{attribute addProperty BoxType "EPP1816-3008-0016"}
{attribute addProperty Id "StatusAT %I*Status_9EB472D91620ValueAT %I*INT16217"}
{attribute addProperty CRC "911372288"}
{attribute addProperty SizeInBites "32"}
{attribute addProperty SizeInBytes "4"}
TYPE AI_Inputs_Channel_36527000 :
STRUCT
	{attribute addProperty Name "Status"}
	Status AT %I* : Status_9EB472D9;
	{attribute addProperty Name "Value"}
	Value AT %I* : INT;
END_STRUCT
END_TYPE

(* stored: Version 1.2.0.0, ProductVersion 3.1.4024.9
   DUT AI_Inputs_Channel_36527000: Id {480c2a12-c070-4b8e-93cb-b691dc561522} *)
